FUNCTION_BLOCK fb_datareturn
VAR_INPUT
	
	ReturnBetweenDates:ST_ReturnBetweenDates;
END_VAR

VAR_OUTPUT
	recordarray: ARRAY [0..1500] OF STRING(100);
	bReady:bool:=false;
END_VAR
VAR
	bExecute:BOOL:=FALSE;
	i:int;
	
END_VAR

METHOD ClearRecordArray : BOOL
VAR_INPUT
END_VAR
i:=0;
FOR i:=0 TO 1500 BY 1 DO
	RecordArray[i]:='';
END_FOR
END_METHOD

METHOD execute : BOOL
VAR_INPUT
END_VAR
bExecute:=TRUE;
END_METHOD

METHOD reset : BOOL
VAR_INPUT
END_VAR
bExecute:=FALSE;


bReady:=false;
END_METHOD

END_FUNCTION_BLOCK

(* stored: Version 1.1.0.1, ProductVersion 3.1.4024.2
   POU fb_datareturn: Id {c100812c-ae12-4014-8498-7296c5fbc1fa}, SpecialFunc None
   Method ClearRecordArray: Id {1e605597-1444-4e9c-9d4b-8ff92b12cca7}
   Method execute: Id {2618e7e0-b2fa-42ab-bc05-fddcb3da03c0}
   Method reset: Id {aa8f61d9-0d8d-42ca-92c7-f44437e7b9bb} *)
